TYPE AxesDialogAlphaUnits :
(
	DIALOG_HMS := 0,
    DIALOG_HOURS := 1,
    DIALOG_RADIANS := 2
);
END_TYPE

(* stored: Version 1.1.0.1, ProductVersion 3.1.4018.5
   DUT AxesDialogAlphaUnits: Id {45acd258-3df6-4db2-830c-ab0a7f3feb7f} *)
